FUNCTION_BLOCK GF_Zirkulieren EXTENDS FB_Basis
VAR_INPUT
	// Instanzieren von Sensoren mit Interfaces
	
	// Instanzieren von Aktoren mit Interfaces
	Ventil_IN			:I_Magnetventil;
	Ventil_OUT			:I_Magnetventil;
	
	Pumpe				:I_Motor2R;
	
END_VAR
VAR_OUTPUT
	
END_VAR
VAR
	
END_VAR

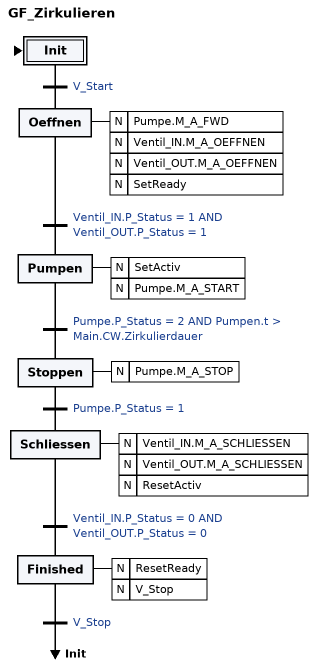
INITIAL_STEP Init:
END_STEP
TRANSITION FROM Init TO Oeffnen
    := V_Start;
END_TRANSITION
STEP Oeffnen:
    Pumpe.M_A_FWD(N);
    Ventil_IN.M_A_OEFFNEN(N);
    Ventil_OUT.M_A_OEFFNEN(N);
    SetReady(N);
END_STEP
TRANSITION FROM Oeffnen TO Pumpen
    := Ventil_IN.P_Status = 1 AND Ventil_OUT.P_Status = 1;
END_TRANSITION
STEP Pumpen:
    SetActiv(N);
    Pumpe.M_A_START(N);
END_STEP
TRANSITION FROM Pumpen TO Stoppen
    := Pumpe.P_Status = 2 AND Pumpen.t > Main.CW.Zirkulierdauer;
END_TRANSITION
STEP Stoppen:
    Pumpe.M_A_STOP(N);
END_STEP
TRANSITION FROM Stoppen TO Schliessen
    := Pumpe.P_Status = 1;
END_TRANSITION
STEP Schliessen:
    Ventil_IN.M_A_SCHLIESSEN(N);
    Ventil_OUT.M_A_SCHLIESSEN(N);
    ResetActiv(N);
END_STEP
TRANSITION FROM Schliessen TO Finished
    := Ventil_IN.P_Status = 0 AND Ventil_OUT.P_Status = 0;
END_TRANSITION
STEP Finished:
    ResetReady(N);
    V_Stop(N);
END_STEP
TRANSITION FROM Finished TO Init
    := V_Stop;
END_TRANSITION

ACTION ResetActiv:
MAIN.SW.PrimActiv := FALSE;
END_ACTION

ACTION ResetReady:
MAIN.SW.PrimReady := FALSE;
END_ACTION

ACTION SetActiv:
MAIN.SW.PrimActiv := TRUE;
END_ACTION

ACTION SetReady:
MAIN.SW.PrimReady := TRUE;
END_ACTION

END_FUNCTION_BLOCK

(* stored: Version 1.1.0.1, ProductVersion 3.1.4024.12
   POU GF_Zirkulieren: Id {a3450a1b-12e1-4c04-8ad2-9bb2cd306dac}, SpecialFunc None
   Folder 01_Aktionen: Id {b286a800-5ca6-40dc-994e-348370a92f4c}
   Action ResetActiv: Id {b6be454c-8fc4-4f05-89e0-add6a3aa6f6a}
   Action ResetReady: Id {88d86819-d352-4c00-8bf7-b519139799f4}
   Action SetActiv: Id {5f4ab24d-23e3-476d-9ced-7224ca24c7fc}
   Action SetReady: Id {9b1208bb-c542-492d-887a-784a4b6b989d} *)
